(* CoDeSys 2.3 project: TTC_test.pro *)
(* Libraries: cl_base.lib 7.7.15 13:13:12, TTControl.lib 12.3.09 20:55:14, Standard.lib 12.3.09 20:55:14, lib60.lib 24.1.18 21:39:36, lib60_data_types.lib 23.1.18 21:22:42 *)

(* PLC configuration (modules and I/O channels)
ADC_5V Mode configured by SW [ADC_5V] node 0, in %IB0 out %QB0
  Not used [not_used] node 0, in %IB0 out %QB0
  Not used [not_used] node 1, in %IB0 out %QB0
  Not used [not_used] node 2, in %IB0 out %QB0
  Not used [not_used] node 3, in %IB0 out %QB0
  Not used [not_used] node 4, in %IB0 out %QB0
  Not used [not_used] node 5, in %IB0 out %QB0
  Not used [not_used] node 6, in %IB0 out %QB0
  Not used [not_used] node 7, in %IB0 out %QB0
ADC_32V range configured by SW [ADC_Range_by_SW] node 1, in %IB0 out %QB0 {ADC_Range = 0-32V; ADC_Range = 0-5V}
  Not used [not_used] node 0, in %IB0 out %QB0
  Not used [not_used] node 1, in %IB0 out %QB0
  Not used [not_used] node 2, in %IB0 out %QB0
  Not used [not_used] node 3, in %IB0 out %QB0
  Not used [not_used] node 4, in %IB0 out %QB0
  Not used [not_used] node 5, in %IB0 out %QB0
  Not used [not_used] node 6, in %IB0 out %QB0
  Not used [not_used] node 7, in %IB0 out %QB0
CURRENT_MEASURE AT %IW0 [WordInput] mA
PWMCM_0_stat AT %IW2 [WordInput]
Not used [not_used] node 1, in %IB4 out %QB0
Not used [not_used] node 2, in %IB4 out %QB0
Not used [not_used] node 3, in %IB4 out %QB0
ENCODER AT %IW4 [WordInput]
TI_8_stat AT %IW6 [WordInput]
TI 9 (INC secondary) [TI_Incremental_1] node 1, in %IB8 out %QB0
Not used [not_used] node 2, in %IB8 out %QB0
Not used [not_used] node 3, in %IB8 out %QB0
DigIN [Dig_IN] node 4, in %IB8 out %QB0
  Not used [not_used] node 0, in %IB8 out %QB0
  Not used [not_used] node 1, in %IB8 out %QB0
  Not used [not_used] node 2, in %IB8 out %QB0
  Not used [not_used] node 3, in %IB8 out %QB0
  Not used [not_used] node 4, in %IB8 out %QB0
  Not used [not_used] node 5, in %IB8 out %QB0
  Not used [not_used] node 6, in %IB8 out %QB0
  Not used [not_used] node 7, in %IB8 out %QB0
PROP_VAL AT %QW0 [WordOutput]
PWM_0_duty_fb AT %ID8 [DoubleWordInput]
PWM_0_stat AT %IW12 [WordInput]
Not used [not_used] node 1, in %IB14 out %QB2
Not used [not_used] node 2, in %IB14 out %QB2
Not used [not_used] node 3, in %IB14 out %QB2
Not used [not_used] node 4, in %IB14 out %QB2
Not used [not_used] node 5, in %IB14 out %QB2
Not used [not_used] node 6, in %IB14 out %QB2
Not used [not_used] node 7, in %IB14 out %QB2
DigOUT or AnalogIN [DigOUT_or_AnIN] node 6, in %IB14 out %QB2
  Not used [not_used] node 0, in %IB14 out %QB2
  Not used [not_used] node 1, in %IB14 out %QB2
  Not used [not_used] node 2, in %IB14 out %QB2
  Not used [not_used] node 3, in %IB14 out %QB2
  Not used [not_used] node 4, in %IB14 out %QB2
  Not used [not_used] node 5, in %IB14 out %QB2
  Not used [not_used] node 6, in %IB14 out %QB2
  Not used [not_used] node 7, in %IB14 out %QB2
Interfaces [INTERFAC] node 7, in %IB14 out %QB2
  Not used [not_used] node 0, in %IB14 out %QB2
  Not used [not_used] node 1, in %IB14 out %QB2
  CAN 1 [IO_CAN_CHANNEL_1] node 3, in %IB14 out %QB2 {CAN_Baudrate = 500 kb/s; CAN_Tseg1 = 5; CAN_Tseg2 = 3; CAN_Sjw = 2}
Generic Functions [GENERIC] node 8, in %IB14 out %QB2
  Retain_stat AT %IW14 [WordInput]
  PWM_Enable AT %QB2 [BoolOutput]
  Sleep_Mode AT %QB4 [BoolOutput]
  K15 [K15] node 0, in %IB16 out %QB6
    K15_val AT %IB16 [BoolInput]
    K15_stat AT %IW18 [WordInput]
  Sensor Supply 5V 0 [UGEB0] node 1, in %IB20 out %QB6 {SensSup = ENABLE; BoolType = DISABLE}
    SS0_val AT %IW20 [WordInput] mV
    SS0_fresh AT %IB22 [BoolInput]
    SS0_stat AT %IW24 [WordInput]
  Sensor Supply 5V 1 [UGEB1] node 2, in %IB26 out %QB6 {SensSup = ENABLE; BoolType = DISABLE}
    SS1_val AT %IW26 [WordInput] mV
    SS1_fresh AT %IB28 [BoolInput]
    SS1_stat AT %IW30 [WordInput]
  Variable Sensor Supply [UGEBVAR] node 3, in %IB32 out %QB6 {VarSens = 8.5 V; BoolType = DISABLE}
    SS_var_val AT %IW32 [WordInput] mV
    SS_var_fresh AT %IB34 [BoolInput]
    SS_var_stat AT %IW36 [WordInput]
  Board Temperature [BOARDTEMP] node 4, in %IB38 out %QB6 {BoolType = DISABLE}
    Board_temp_val AT %ID38 [RealInput] °C
    Board_temp_fresh AT %IB42 [BoolInput]
    Board_temp_stat AT %IW44 [WordInput]
  Battery Voltage [BATTVOLT] node 5, in %IB46 out %QB6
    Battery_val AT %IW46 [WordInput] mV
    Battery_fresh AT %IB48 [BoolInput]
    Battery_stat AT %IW50 [WordInput]
  Cycle Load Statistics [CYCLELOAD] node 6, in %IB52 out %QB6
    CycleLoad AT %ID52 [DoubleWordInput] us
    CycleLoadMin AT %ID56 [DoubleWordInput] us
    CycleLoadMax AT %ID60 [DoubleWordInput] us
    ResetLoadStat AT %QB6 [BoolOutput]
*)

(* Global variable list: Global_Variables *)
VAR_GLOBAL CONSTANT
	CAN_MAX_TX_BUF: BYTE := 10;
	CAN_MAX_RX_BUF: BYTE := 10;
END_VAR
VAR_GLOBAL
	gCan1          : tCan;                  (* Structure for sending / receiving CAN messages *)
END_VAR

(* Data type *)
TYPE tCan :
STRUCT
	hReceiver: ARRAY [0..CAN_MAX_RX_BUF] OF BYTE;
	hTransmitter: ARRAY [0..CAN_MAX_TX_BUF] OF BYTE;
	Channel: BYTE;
	CanMsg: tCanMsg;
	EcuCycleTime: TIME;
	cReceiverCnt: UINT;
	cTransmitterCnt: UINT;
END_STRUCT
END_TYPE

(* Data type *)
TYPE tCanMsg :
STRUCT
	Data: ARRAY[0..7] OF BYTE;
	CobId: UDINT;
	Length: BYTE;
	Id_Format: BYTE;
END_STRUCT
END_TYPE

(* POU PLC_PRG, FBD *)
PROGRAM PLC_PRG
VAR
END_VAR
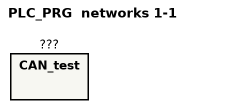
_FBD_ (* Function Block Diagram *)
NETWORK 1
	???:CAN_test()
_END_FBD_
END_PROGRAM

(* POU CAN_test, LD *)
PROGRAM CAN_test
VAR
	Rx_100: CanRx;
	Tx_200: CanTx;
	DATA: ARRAY [0..7] OF BYTE := 16#AA, 16#BB, 16#CC, 16#DD, 16#EE, 16#FF, 16#44, 16#55;
	WORD1: WORD;
	WORD2: WORD;
	V1: WORD;
	V2: WORD;

	X: INT;
	Y: INT;
	Rx_234: CanRx;
	WORD3: WORD;
	WORD4: WORD;
	X1: INT;
	Y1: INT;
	X2: INT;
	Y2: INT;
	a: INT := 5;
	B: INT := 5;
	V: INT;
END_VAR
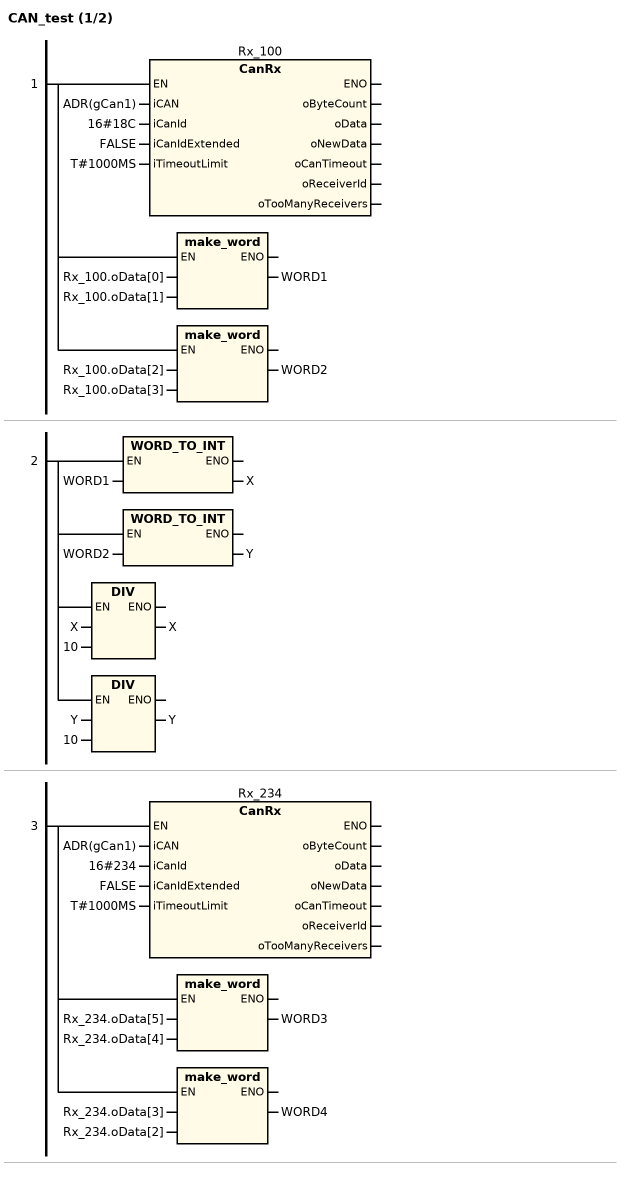
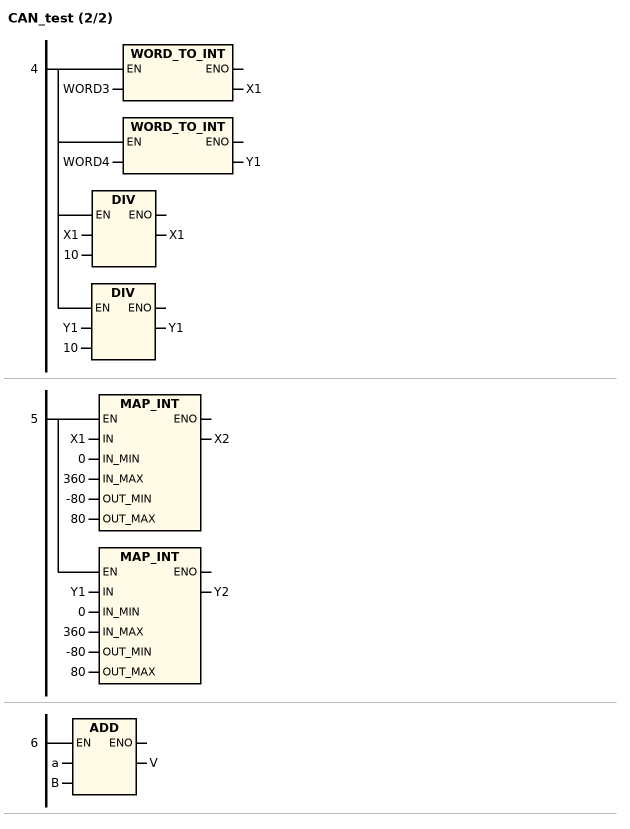
_LD_ (* Ladder Diagram *)
NETWORK 1
	*
		EN --- Rx_100:CanRx(iCAN: ADR(gCan1), iCanId: 16#18C, iCanIdExtended: FALSE, iTimeoutLimit: T#1000MS)
		EN --- make_word(Rx_100.oData[0], Rx_100.oData[1]) => WORD1
		EN --- make_word(Rx_100.oData[2], Rx_100.oData[3]) => WORD2
NETWORK 2
	*
		EN --- WORD_TO_INT(WORD1) => X
		EN --- WORD_TO_INT(WORD2) => Y
		EN --- DIV(X, 10) => X
		EN --- DIV(Y, 10) => Y
NETWORK 3
	*
		EN --- Rx_234:CanRx(iCAN: ADR(gCan1), iCanId: 16#234, iCanIdExtended: FALSE, iTimeoutLimit: T#1000MS)
		EN --- make_word(Rx_234.oData[5], Rx_234.oData[4]) => WORD3
		EN --- make_word(Rx_234.oData[3], Rx_234.oData[2]) => WORD4
NETWORK 4
	*
		EN --- WORD_TO_INT(WORD3) => X1
		EN --- WORD_TO_INT(WORD4) => Y1
		EN --- DIV(X1, 10) => X1
		EN --- DIV(Y1, 10) => Y1
NETWORK 5
	*
		EN --- MAP_INT(IN: X1, IN_MIN: 0, IN_MAX: 360, OUT_MIN: -80, OUT_MAX: 80) => X2
		EN --- MAP_INT(IN: Y1, IN_MIN: 0, IN_MAX: 360, OUT_MIN: -80, OUT_MAX: 80) => Y2
NETWORK 6
	*
		EN --- ADD(a, B) => V
_END_LD_
(* the same logic as Structured Text *)
(* Network 1 *)
Rx_100(iCAN := ADR(gCan1), iCanId := 16#18C, iCanIdExtended := FALSE, iTimeoutLimit := T#1000MS);
WORD1 := make_word(Rx_100.oData[0], Rx_100.oData[1]);
WORD2 := make_word(Rx_100.oData[2], Rx_100.oData[3]);
(* Network 2 *)
X := WORD_TO_INT(WORD1);
Y := WORD_TO_INT(WORD2);
X := X / 10;
Y := Y / 10;
(* Network 3 *)
Rx_234(iCAN := ADR(gCan1), iCanId := 16#234, iCanIdExtended := FALSE, iTimeoutLimit := T#1000MS);
WORD3 := make_word(Rx_234.oData[5], Rx_234.oData[4]);
WORD4 := make_word(Rx_234.oData[3], Rx_234.oData[2]);
(* Network 4 *)
X1 := WORD_TO_INT(WORD3);
Y1 := WORD_TO_INT(WORD4);
X1 := X1 / 10;
Y1 := Y1 / 10;
(* Network 5 *)
X2 := MAP_INT(IN := X1, IN_MIN := 0, IN_MAX := 360, OUT_MIN := -80, OUT_MAX := 80);
Y2 := MAP_INT(IN := Y1, IN_MIN := 0, IN_MAX := 360, OUT_MIN := -80, OUT_MAX := 80);
(* Network 6 *)
V := a + B;
END_PROGRAM

(* POU CAN/CAN2_0b/CanRx, ST *)
(*******************************************************************************
*  Copyright (C) 2011 TTControl S.r.l. All rights reserved.
*  Via Julius Durst 66, I-39042 Bressanone (BZ), Italy, office@ttcontrol.com
*
*  PRE: 			none 
*  POST: 			none
*  GLOBAL:			gCan
*  LIBRARIES:		lib60.lib
*  DESCRIPTION: 	This POU is a high level function block to receive a single CAN-message (the newest one). 
*					
*  REVISION HISTORY:	
*  2013-10-01	joh		Creation
*  2013-11-26	kkh		some comments added/updated, name of global CAN message variable changed to gCan, updated to fullfill latest Coding Guidelines
*  2015-11-11   joh		Fixing issue87479.
*
*******************************************************************************)
FUNCTION_BLOCK CanRx
VAR_INPUT
	iCAN			: POINTER TO tCAN;
	iCanId			: UDINT; 			(* CAN Id *)
	iCanIdExtended	: BOOL; 			(* FALSE = 11-bit, TRUE = 29-bit *)
	iTimeoutLimit	: TIME; 			(* if the specified PGN is not received within ui16TimeoutLimit ms, output bJ1939Timeout is TRUE *)
END_VAR
VAR_OUTPUT
	oByteCount			: BYTE; 				(* number of bytes received *)
	oData				: ARRAY [0..7] OF BYTE; (* data received *)
	oNewData			: BOOL; 				(* flag IF new data has been received *)
	oCanTimeout			: BOOL; 				(* TRUE if timeout has reached. see ui16TimeoutLimit *)
	oReceiverId			: UINT := 65535; 		(* unique receiver ID for internal CAN management *)
	oTooManyReceivers	: BOOL := FALSE; 		(* if TRUE the number of defined receiver FB exceeds CAN_MAX_RX_BUF -> message is not setup - received *)
END_VAR
VAR
	fbCanRx				: RxBufferCan;			(* function block that handles the low level recieve *)
	Timeout				: BOOL;					(* Timeout flag *)
	Init				: BOOL := FALSE;		(* local variable for initializing on first cycle *)
	TempVar				: DWORD;				(* temporary variable *)
	fbTimeOutTon		: TON;					(* Timeout timer *)
	Result				: WORD;					(* Error code from library function calls *)
END_VAR
IF iCAN <> 0 THEN

	(* do an initialization of receiver id with the first call of this function block and
	   check if receiver id is within limit CAN_RX_MESSAGE_NUMBER.
	   Do also an initialization OF RX message buffer with the appropriate mask *)
	IF Init = FALSE THEN
		IF iCAN^.cReceiverCnt <= CAN_MAX_RX_BUF THEN
			(* configure CAN buffer *)
			Result := xc_can_config_msg(ADR(iCAN^.hReceiver[iCAN^.cReceiverCnt]), iCAN^.Channel, 1, IO_CAN_MSG_READ, BOOL_TO_BYTE(iCanIdExtended), iCanId, 16#1FFFFFFF);
			(* increase receiver id *)
			oReceiverId := iCAN^.cReceiverCnt;
			iCAN^.cReceiverCnt := iCAN^.cReceiverCnt + 1;
			IF (iCAN^.cReceiverCnt > CAN_MAX_RX_BUF) OR (Result <> IO_E_OK) THEN
				oTooManyReceivers := TRUE;
			END_IF	(* ELSE do nothing *)
		ELSE
			oTooManyReceivers := TRUE;
		END_IF
		Init := TRUE;
	ELSE
		(* if buffer has been initialiazed and number of receiver is OK, CAN messages are read *)
		IF (Init = TRUE) AND (oReceiverId <> 65535) AND (oTooManyReceivers = FALSE) THEN

			(* read J1939 message *)
			fbCanRx(	iCAN:=iCAN,
						iMsgBuffer := oReceiverId,
						iEnable:=TRUE,
						oNewData=>);

			oNewData := fbCanRx.oNewData;

			(* new data has been received -> save data and necessary output informations *)
			IF oNewData THEN
				oData := iCAN^.CanMsg.Data;
				oByteCount := iCAN^.CanMsg.Length;
				timeout := FALSE;
			END_IF	(* ELSE do nothing *)
	
			(* Check for timeout *)
			fbTimeOutTon(IN:= oNewData = FALSE, PT:= iTimeoutLimit, Q=> Timeout, ET=> );

			oCanTimeout := timeout;
		ELSE
			(* reset outputs *)
			oNewData := FALSE;
			oCanTimeout := TRUE;
			oByteCount := 0;
		END_IF
	END_IF
ELSE
	oNewData := FALSE;
	oCanTimeout := TRUE;
	oByteCount := 0;
END_IF
END_FUNCTION_BLOCK

(* POU CAN/CAN_Low_Level/RxBufferCan, ST *)
(*******************************************************************************
* Copyright (C) 2014 TTControl S.r.l. All rights reserved.
* Via Julius Durst 66, I-39042 Bressanone (BZ), Italy, office@ttcontrol.com
*
* PRE: -
* POST: -
* GLOBAL: -
* LIBRARIES lib94.lib
* DESCRIPTION: Function Block to read a Can Buffer
* REVISION HISTORY:
*
* 2014-07-01  JOH       creation
* 2015-11-11  JOH		Fixing issue87479.
*
*******************************************************************************)
FUNCTION_BLOCK RxBufferCan
VAR_INPUT
	iCAN		: POINTER TO tCan;
	iMsgBuffer  : UINT;
	iEnable		: BOOL;			(* Enable of FB *)
END_VAR
VAR_OUTPUT
	oNewData	: BOOL;			(* new data flag *)
END_VAR
VAR
	ResCanRead	: WORD;			(* return value of CAN read *)
	NrMsgRead	: BYTE;			(* number of read CAN frames *)
	CanData		: t_can_frame;	(* CAN frame *)
	i			: BYTE;
END_VAR
IF iCAN <> 0 THEN

	IF ((iEnable = TRUE) AND (iMsgBuffer <= CAN_MAX_RX_BUF)) THEN
		(* Reset new data flag *)
		oNewData := FALSE;
		(* Call low I/O Driver can read function *)
		ResCanRead := xc_can_read (iCAN^.hReceiver[iMsgBuffer], ADR(CanData), 1, ADR(NrMsgRead));
	
		IF (ResCanRead = IO_E_OK) OR (ResCanRead = IO_E_CAN_OVERFLOW) THEN
			(* Read was succesully *)
			FOR i := 0 TO 7 DO
				(* Copy CAN data *)
				iCAN^.CanMsg.Data[i] := CanData.data[i];
			END_FOR
			(* Copy CAN frame information *)
			iCAN^.CanMsg.CobId := CanData.id;
			iCAN^.CanMsg.Id_Format := CanData.id_format;
			iCAN^.CanMsg.Length := CanData.length;
			(* Set new data flag *)
			oNewData := TRUE;
		END_IF	(* ELSE do nothing *)

	ELSE

		(* reset variables *)
		oNewData := FALSE;

	END_IF	(* ELSE do nothing *)

ELSE

	(* reset variables *)
	oNewData := FALSE;

END_IF
END_FUNCTION_BLOCK

(* POU CAN/CAN2_0b/CanTx, ST *)
(*******************************************************************************
*  Copyright (C) 2011 TTControl S.r.l. All rights reserved.
*  Via Julius Durst 66, I-39042 Bressanone (BZ), Italy, office@ttcontrol.com
*
*  PRE: 			none 
*  POST: 			none
*  GLOBAL:			gCan
*  LIBRARIES:		lib60.lib
*  DESCRIPTION: 	This POU is a high level function block to transmit CAN-messages. 
*					
*  REVISION HISTORY:	
*  2013-10-01	joh		Creation
*  2013-11-26	kkh		some comments added/updated, name of global CAN message variable changed to gCan, update to fullfill latest Coding Guidelines
*  2014-07-25   joh		Added iForceSend .
*  2015-11-11   joh		Fixing issue87479.
*
*******************************************************************************)
FUNCTION_BLOCK CanTx
VAR_INPUT
	iEnable			: BOOL;					(* enables sending of message *)
	iCAN			: POINTER TO tCan;
	iForceSend		: BOOL;					(* force sending independnent of iTransmitRate *)
	iTransmitRate	: TIME; 				(* transmit rate of function block *)
	iCanId			: UDINT; 				(* CAN ID *)
	iCanIdExtended	: BOOL; 				(* FALSE = 11-bit, TRUE = 29-bit *)
	iByteCount		: BYTE; 				(* number of bytes to transmit *)
	iData			: ARRAY [0..7] OF BYTE; (* data to transmit *)
END_VAR
VAR_OUTPUT
	oTransmitterId		: UINT := 65535; (* unique transmitter ID for internal CAN management *)
	oTooManyTransmitters: BOOL := FALSE; (* if TRUE the number of defined transmitter FB exceeds CAN_MAX_TX_BUF -> message is not setup - transmitted  *)
	oMsgSent			: BOOL := FALSE; (* TRUE: message has been sent, FALSE: message has not been sent *)
END_VAR
VAR
	fbCanTx			: TxBufferCan; 		(* function block that handles the low level transmission *)
	InitMessage		: BOOL := FALSE; 	(* local variable for initializing on first cycle *)
	fbTonTransmit	: TON; 				(* timer for transmit rate *)
	FirstCycle		: BOOL := TRUE;		(* send in the first cycle *)
	CanHandle		: BYTE;
	Result			: WORD;				(* Error code from library function calls *)
END_VAR
IF iCAN <> 0 THEN
	IF iEnable THEN
	
		(* do an initialization of transmitter id with the first call of this function block and
		   check if transmitter id is within LIMIT CAN_TX_MESSAGE_NUMBER *)
		IF InitMessage = FALSE THEN
			IF iCAN^.cTransmitterCnt  <= CAN_MAX_TX_BUF THEN
				(* configure CAN buffer *)
				xc_can_config_msg(ADR(iCan^.hTransmitter[iCan^.cTransmitterCnt]), iCan^.Channel, 1, IO_CAN_MSG_WRITE, BOOL_TO_BYTE(iCanIdExtended), 0, 0);
				oTransmitterId := iCan^.cTransmitterCnt;
				iCan^.cTransmitterCnt := oTransmitterId + 1;
				IF (iCan^.cTransmitterCnt > CAN_MAX_TX_BUF) OR (Result <> IO_E_OK) THEN
					oTooManyTransmitters := TRUE;
				END_IF
			ELSE
				oTooManyTransmitters := TRUE;
			END_IF
			InitMessage := TRUE;
			oMsgSent := FALSE;
	
		ELSE
		
			(* if iForceSend is TRUE, then the transmit timer is resetted, Msg should be send immediately *)
			IF NOT(iForceSend) THEN
				fbTonTransmit(	IN := iEnable,
								PT := iTransmitRate - iCan^.EcuCycleTime);
			ELSE
				fbTonTransmit( 	IN := FALSE);
			END_IF
	
			(* message is send if the timer is passed or message should be sent now or at the very first cycle *)
			IF fbTonTransmit.Q OR iForceSend OR FirstCycle THEN
				(* reset timer *)
				fbTonTransmit(IN := FALSE);
				(* do process only if it is a valid transmitter id -> bTooManyTransmitters = FALSE *)
				IF (oTooManyTransmitters = FALSE) THEN
					(* check valid range for ui8ByteCount *)
					IF (iByteCount > 8) THEN
						iByteCount := 8;
					END_IF
	
					(* send CAN message *)
					fbCanTx(	iCan := iCan,
								iMsgId:= iCanId,
								iExtendedId:= iCanIdExtended,
								iData:= iData,
								iTransmitterId := oTransmitterId,
								iLength:= iByteCount,
								iEnable:= TRUE);
				ELSE
					oMsgSent := FALSE;
				END_IF
				FirstCycle := FALSE;
			ELSE
				oMsgSent := FALSE;
			END_IF
		END_IF 
	ELSE
		(* reset timer *)
		fbTonTransmit( IN := FALSE);
		FirstCycle := TRUE;	
		oMsgSent := FALSE;
	END_IF
ELSE
	(* reset timer *)
	fbTonTransmit( IN := FALSE);
	FirstCycle := TRUE;	
	oMsgSent := FALSE;
END_IF
END_FUNCTION_BLOCK

(* POU CAN/CAN_Low_Level/TxBufferCan, ST *)
(*******************************************************************************
* Copyright (C) 2014 TTControl S.r.l. All rights reserved.
* Via Julius Durst 66, I-39042 Bressanone (BZ), Italy, office@ttcontrol.com
*
* PRE: -
* POST: -
* GLOBAL: -
* LIBRARIES lib94.lib
* DESCRIPTION: Function Block to write a Can Buffer
* REVISION HISTORY:
*
* 2014-07-01  JOH       creation
*
*******************************************************************************)
FUNCTION_BLOCK TxBufferCan
VAR_INPUT
	iCAN		: POINTER TO tCAN;
	iMsgId		: UDINT;	(* CAN Id *)
	iExtendedId	: BOOL;		(* Flag Id is a Standard 11-bit or an Extended 29-bit*)
	iData		: ARRAY[0..7] OF BYTE;
	iTransmitterId: UINT;
	iLength		: BYTE;		(* Length of data frame *)
	iEnable		: BOOL;		(* Enable of FB *)
END_VAR
VAR_OUTPUT
	oMsgSent	: BOOL;
END_VAR
VAR
	ResCanWrite	: WORD;		(* return value of CAN read *)
	CanData		: t_can_frame;
	i			: BYTE;
END_VAR
IF iCAN <> 0 THEN
	IF (iEnable = TRUE) AND (iLength >= 1) AND (iLength <= 8) THEN
	
		(* prepare data *)
		FOR i := 0 TO (iLength - 1) BY 1 DO
			CanData.data[i] := iData[i];
		END_FOR

		CanData.id := iMsgId;
		CanData.id_format := BOOL_TO_BYTE(iExtendedId);
		CanData.length := iLength;
	
		(* send data *)
		ResCanWrite := xc_can_write (iCAN^.hTransmitter[iTransmitterId], ADR(CanData), 1);
		IF (ResCanWrite = IO_E_OK) THEN
			oMsgSent := TRUE;
		ELSE
			oMsgSent := FALSE;
		END_IF

	ELSE
		oMsgSent := FALSE;
	END_IF
ELSE
	oMsgSent := FALSE;
END_IF
END_FUNCTION_BLOCK

(* POU FB_LIBRARY/MAP_INT, ST *)
FUNCTION MAP_INT : INT
(*
Author: Nikshitha S
Date: 10-08-2023
Description: This particular function works on inputs and outputs both with INTEGER datatype. Thus consuming less memory.
*)
VAR_INPUT
	IN: INT;
	IN_MIN:INT;
	IN_MAX : INT;
	OUT_MIN:INT;
	OUT_MAX:INT;
END_VAR

VAR
	ERROR: BOOL;
	FINAL_MAP: INT;
	INPUT_RANGE: INT;
	OUTPUT_RANGE: INT;
END_VAR
ERROR := (IN_MAX-IN_MIN=0) OR (IN<IN_MIN) OR (IN>IN_MAX);

INPUT_RANGE := IN_MAX-IN_MIN;
OUTPUT_RANGE := OUT_MAX-OUT_MIN;

MAP_INT:= ((IN-IN_MIN)*OUTPUT_RANGE) / INPUT_RANGE + OUT_MIN;


IF ERROR AND (IN<IN_MIN)THEN
MAP_INT:=OUT_MIN;
END_IF

IF ERROR AND (IN>IN_MAX)THEN
MAP_INT:=OUT_MAX;
END_IF
END_FUNCTION

(* POU CAN/CanInit, ST *)
PROGRAM CanInit
VAR_INPUT
	iEnable 		: BOOL;				(* enable initialization flag *)
	iChannel		: BYTE; 			(* CAN channel 0 ... x *)
	iCAN			: POINTER TO tCan; 	(* pointer to CAN structure *)
	iEcuCycleTime	: TIME; 			(* cycle time of task calling can transmit and receive FB *)
END_VAR
IF iCan <> 0 THEN
	(* initialize the CAN *)
	IF iEnable THEN
		iCAN^.EcuCycleTime := iEcuCycleTime;
		iCAN^.Channel := iChannel;
		iCAN^.cReceiverCnt := 0;
		iCAN^.cTransmitterCnt := 0;
	END_IF
END_IF
END_PROGRAM

(* POU rot_enc, LD *)
PROGRAM rot_enc
VAR_INPUT
END_VAR
VAR_OUTPUT
END_VAR
VAR
END_VAR
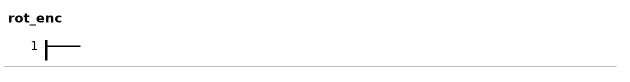
_LD_ (* Ladder Diagram *)
NETWORK 1
	*
_END_LD_
(* the same logic as Structured Text *)
(* Network 1 *)
END_PROGRAM

(* POU TEST_ANALOG, LD *)
 PROGRAM TEST_ANALOG
VAR
END_VAR
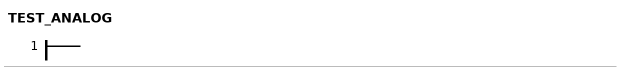
_LD_ (* Ladder Diagram *)
NETWORK 1
	*
_END_LD_
(* the same logic as Structured Text *)
(* Network 1 *)
END_PROGRAM

(* POU TEST_DIG, LD *)
PROGRAM TEST_DIG
VAR
END_VAR
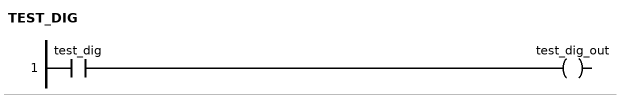
_LD_ (* Ladder Diagram *)
NETWORK 1
	[test_dig] --- (test_dig_out)
_END_LD_
(* the same logic as Structured Text *)
(* Network 1 *)
test_dig_out := test_dig;
END_PROGRAM
